{attribute 'GeneratedUsingTerminal: KL6211-0004'}
{attribute addProperty BoxType "KL6211-0004"}
{attribute addProperty Id "StatusAT %I*UINT0Parameter_InAT %I*UDINT0ASI_In_Slave_1_StatusAT %I*USINT0ASI_In_Slave_3_Slave_2AT %I*USINT0ASI_In_Slave_5_Slave_4AT %I*USINT0ASI_In_Slave_7_Slave_6AT %I*USINT0ASI_In_Slave_9_Slave_8AT %I*USINT0ASI_In_Slave_11_Slave_10AT %I*USINT0ASI_In_Slave_13_Slave_12AT %I*USINT0ASI_In_Slave_15_Slave_14AT %I*USINT0ASI_In_Slave_17_Slave_16AT %I*USINT0ASI_In_Slave_19_Slave_18AT %I*USINT0ASI_In_Slave_21_Slave_20AT %I*USINT0ASI_In_Slave_23_Slave_22AT %I*USINT0ASI_In_Slave_25_Slave_24AT %I*USINT0ASI_In_Slave_27_Slave_26AT %I*USINT0ASI_In_Slave_29_Slave_28AT %I*USINT0ASI_In_Slave_31_Slave_30AT %I*USINT0ASI_In_Slave_33_Slave_32AT %I*USINT0ASI_In_Slave_35_Slave_34AT %I*USINT0ASI_In_Slave_37_Slave_36AT %I*USINT0ASI_In_Slave_39_Slave_38AT %I*USINT0ASI_In_Slave_41_Slave_40AT %I*USINT0ASI_In_Slave_43_Slave_42AT %I*USINT0ASI_In_Slave_45_Slave_44AT %I*USINT0ASI_In_Slave_47_Slave_46AT %I*USINT0ASI_In_Slave_49_Slave_48AT %I*USINT0ASI_In_Slave_51_Slave_50AT %I*USINT0ASI_In_Slave_53_Slave_52AT %I*USINT0ASI_In_Slave_55_Slave_54AT %I*USINT0ASI_In_Slave_57_Slave_56AT %I*USINT0ASI_In_Slave_59_Slave_58AT %I*USINT0ASI_In_Slave_61_Slave_60AT %I*USINT0ASI_In_Slave_63_Slave_62AT %I*USINT0ControlAT %Q*UINT0Parameter_OutAT %Q*UDINT0ASI_Out_Slave_1_ControlAT %Q*USINT0ASI_Out_Slave_3_Slave_2AT %Q*USINT0ASI_Out_Slave_5_Slave_4AT %Q*USINT0ASI_Out_Slave_7_Slave_6AT %Q*USINT0ASI_Out_Slave_9_Slave_8AT %Q*USINT0ASI_Out_Slave_11_Slave_10AT %Q*USINT0ASI_Out_Slave_13_Slave_12AT %Q*USINT0ASI_Out_Slave_15_Slave_14AT %Q*USINT0ASI_Out_Slave_17_Slave_16AT %Q*USINT0ASI_Out_Slave_19_Slave_18AT %Q*USINT0ASI_Out_Slave_21_Slave_20AT %Q*USINT0ASI_Out_Slave_23_Slave_22AT %Q*USINT0ASI_Out_Slave_25_Slave_24AT %Q*USINT0ASI_Out_Slave_27_Slave_26AT %Q*USINT0ASI_Out_Slave_29_Slave_28AT %Q*USINT0ASI_Out_Slave_31_Slave_30AT %Q*USINT0ASI_Out_Slave_33_Slave_32AT %Q*USINT0ASI_Out_Slave_35_Slave_34AT %Q*USINT0ASI_Out_Slave_37_Slave_36AT %Q*USINT0ASI_Out_Slave_39_Slave_38AT %Q*USINT0ASI_Out_Slave_41_Slave_40AT %Q*USINT0ASI_Out_Slave_43_Slave_42AT %Q*USINT0ASI_Out_Slave_45_Slave_44AT %Q*USINT0ASI_Out_Slave_47_Slave_46AT %Q*USINT0ASI_Out_Slave_49_Slave_48AT %Q*USINT0ASI_Out_Slave_51_Slave_50AT %Q*USINT0ASI_Out_Slave_53_Slave_52AT %Q*USINT0ASI_Out_Slave_55_Slave_54AT %Q*USINT0ASI_Out_Slave_57_Slave_56AT %Q*USINT0ASI_Out_Slave_59_Slave_58AT %Q*USINT0ASI_Out_Slave_61_Slave_60AT %Q*USINT0ASI_Out_Slave_63_Slave_62AT %Q*USINT0"}
{attribute addProperty CRC "2796071749"}
{attribute addProperty Size "0"}
TYPE Channel_A6A8AB45 :
STRUCT
	{attribute addProperty Name "Status"}
	Status AT %I* : UINT;
	{attribute addProperty Name "Parameter_In"}
	Parameter_In AT %I* : UDINT;
	{attribute addProperty Name "ASI_In_Slave_1_Status"}
	ASI_In_Slave_1_Status AT %I* : USINT;
	{attribute addProperty Name "ASI_In_Slave_3_Slave_2"}
	ASI_In_Slave_3_Slave_2 AT %I* : USINT;
	{attribute addProperty Name "ASI_In_Slave_5_Slave_4"}
	ASI_In_Slave_5_Slave_4 AT %I* : USINT;
	{attribute addProperty Name "ASI_In_Slave_7_Slave_6"}
	ASI_In_Slave_7_Slave_6 AT %I* : USINT;
	{attribute addProperty Name "ASI_In_Slave_9_Slave_8"}
	ASI_In_Slave_9_Slave_8 AT %I* : USINT;
	{attribute addProperty Name "ASI_In_Slave_11_Slave_10"}
	ASI_In_Slave_11_Slave_10 AT %I* : USINT;
	{attribute addProperty Name "ASI_In_Slave_13_Slave_12"}
	ASI_In_Slave_13_Slave_12 AT %I* : USINT;
	{attribute addProperty Name "ASI_In_Slave_15_Slave_14"}
	ASI_In_Slave_15_Slave_14 AT %I* : USINT;
	{attribute addProperty Name "ASI_In_Slave_17_Slave_16"}
	ASI_In_Slave_17_Slave_16 AT %I* : USINT;
	{attribute addProperty Name "ASI_In_Slave_19_Slave_18"}
	ASI_In_Slave_19_Slave_18 AT %I* : USINT;
	{attribute addProperty Name "ASI_In_Slave_21_Slave_20"}
	ASI_In_Slave_21_Slave_20 AT %I* : USINT;
	{attribute addProperty Name "ASI_In_Slave_23_Slave_22"}
	ASI_In_Slave_23_Slave_22 AT %I* : USINT;
	{attribute addProperty Name "ASI_In_Slave_25_Slave_24"}
	ASI_In_Slave_25_Slave_24 AT %I* : USINT;
	{attribute addProperty Name "ASI_In_Slave_27_Slave_26"}
	ASI_In_Slave_27_Slave_26 AT %I* : USINT;
	{attribute addProperty Name "ASI_In_Slave_29_Slave_28"}
	ASI_In_Slave_29_Slave_28 AT %I* : USINT;
	{attribute addProperty Name "ASI_In_Slave_31_Slave_30"}
	ASI_In_Slave_31_Slave_30 AT %I* : USINT;
	{attribute addProperty Name "ASI_In_Slave_33_Slave_32"}
	ASI_In_Slave_33_Slave_32 AT %I* : USINT;
	{attribute addProperty Name "ASI_In_Slave_35_Slave_34"}
	ASI_In_Slave_35_Slave_34 AT %I* : USINT;
	{attribute addProperty Name "ASI_In_Slave_37_Slave_36"}
	ASI_In_Slave_37_Slave_36 AT %I* : USINT;
	{attribute addProperty Name "ASI_In_Slave_39_Slave_38"}
	ASI_In_Slave_39_Slave_38 AT %I* : USINT;
	{attribute addProperty Name "ASI_In_Slave_41_Slave_40"}
	ASI_In_Slave_41_Slave_40 AT %I* : USINT;
	{attribute addProperty Name "ASI_In_Slave_43_Slave_42"}
	ASI_In_Slave_43_Slave_42 AT %I* : USINT;
	{attribute addProperty Name "ASI_In_Slave_45_Slave_44"}
	ASI_In_Slave_45_Slave_44 AT %I* : USINT;
	{attribute addProperty Name "ASI_In_Slave_47_Slave_46"}
	ASI_In_Slave_47_Slave_46 AT %I* : USINT;
	{attribute addProperty Name "ASI_In_Slave_49_Slave_48"}
	ASI_In_Slave_49_Slave_48 AT %I* : USINT;
	{attribute addProperty Name "ASI_In_Slave_51_Slave_50"}
	ASI_In_Slave_51_Slave_50 AT %I* : USINT;
	{attribute addProperty Name "ASI_In_Slave_53_Slave_52"}
	ASI_In_Slave_53_Slave_52 AT %I* : USINT;
	{attribute addProperty Name "ASI_In_Slave_55_Slave_54"}
	ASI_In_Slave_55_Slave_54 AT %I* : USINT;
	{attribute addProperty Name "ASI_In_Slave_57_Slave_56"}
	ASI_In_Slave_57_Slave_56 AT %I* : USINT;
	{attribute addProperty Name "ASI_In_Slave_59_Slave_58"}
	ASI_In_Slave_59_Slave_58 AT %I* : USINT;
	{attribute addProperty Name "ASI_In_Slave_61_Slave_60"}
	ASI_In_Slave_61_Slave_60 AT %I* : USINT;
	{attribute addProperty Name "ASI_In_Slave_63_Slave_62"}
	ASI_In_Slave_63_Slave_62 AT %I* : USINT;
	{attribute addProperty Name "Control"}
	Control AT %Q* : UINT;
	{attribute addProperty Name "Parameter_Out"}
	Parameter_Out AT %Q* : UDINT;
	{attribute addProperty Name "ASI_Out_Slave_1_Control"}
	ASI_Out_Slave_1_Control AT %Q* : USINT;
	{attribute addProperty Name "ASI_Out_Slave_3_Slave_2"}
	ASI_Out_Slave_3_Slave_2 AT %Q* : USINT;
	{attribute addProperty Name "ASI_Out_Slave_5_Slave_4"}
	ASI_Out_Slave_5_Slave_4 AT %Q* : USINT;
	{attribute addProperty Name "ASI_Out_Slave_7_Slave_6"}
	ASI_Out_Slave_7_Slave_6 AT %Q* : USINT;
	{attribute addProperty Name "ASI_Out_Slave_9_Slave_8"}
	ASI_Out_Slave_9_Slave_8 AT %Q* : USINT;
	{attribute addProperty Name "ASI_Out_Slave_11_Slave_10"}
	ASI_Out_Slave_11_Slave_10 AT %Q* : USINT;
	{attribute addProperty Name "ASI_Out_Slave_13_Slave_12"}
	ASI_Out_Slave_13_Slave_12 AT %Q* : USINT;
	{attribute addProperty Name "ASI_Out_Slave_15_Slave_14"}
	ASI_Out_Slave_15_Slave_14 AT %Q* : USINT;
	{attribute addProperty Name "ASI_Out_Slave_17_Slave_16"}
	ASI_Out_Slave_17_Slave_16 AT %Q* : USINT;
	{attribute addProperty Name "ASI_Out_Slave_19_Slave_18"}
	ASI_Out_Slave_19_Slave_18 AT %Q* : USINT;
	{attribute addProperty Name "ASI_Out_Slave_21_Slave_20"}
	ASI_Out_Slave_21_Slave_20 AT %Q* : USINT;
	{attribute addProperty Name "ASI_Out_Slave_23_Slave_22"}
	ASI_Out_Slave_23_Slave_22 AT %Q* : USINT;
	{attribute addProperty Name "ASI_Out_Slave_25_Slave_24"}
	ASI_Out_Slave_25_Slave_24 AT %Q* : USINT;
	{attribute addProperty Name "ASI_Out_Slave_27_Slave_26"}
	ASI_Out_Slave_27_Slave_26 AT %Q* : USINT;
	{attribute addProperty Name "ASI_Out_Slave_29_Slave_28"}
	ASI_Out_Slave_29_Slave_28 AT %Q* : USINT;
	{attribute addProperty Name "ASI_Out_Slave_31_Slave_30"}
	ASI_Out_Slave_31_Slave_30 AT %Q* : USINT;
	{attribute addProperty Name "ASI_Out_Slave_33_Slave_32"}
	ASI_Out_Slave_33_Slave_32 AT %Q* : USINT;
	{attribute addProperty Name "ASI_Out_Slave_35_Slave_34"}
	ASI_Out_Slave_35_Slave_34 AT %Q* : USINT;
	{attribute addProperty Name "ASI_Out_Slave_37_Slave_36"}
	ASI_Out_Slave_37_Slave_36 AT %Q* : USINT;
	{attribute addProperty Name "ASI_Out_Slave_39_Slave_38"}
	ASI_Out_Slave_39_Slave_38 AT %Q* : USINT;
	{attribute addProperty Name "ASI_Out_Slave_41_Slave_40"}
	ASI_Out_Slave_41_Slave_40 AT %Q* : USINT;
	{attribute addProperty Name "ASI_Out_Slave_43_Slave_42"}
	ASI_Out_Slave_43_Slave_42 AT %Q* : USINT;
	{attribute addProperty Name "ASI_Out_Slave_45_Slave_44"}
	ASI_Out_Slave_45_Slave_44 AT %Q* : USINT;
	{attribute addProperty Name "ASI_Out_Slave_47_Slave_46"}
	ASI_Out_Slave_47_Slave_46 AT %Q* : USINT;
	{attribute addProperty Name "ASI_Out_Slave_49_Slave_48"}
	ASI_Out_Slave_49_Slave_48 AT %Q* : USINT;
	{attribute addProperty Name "ASI_Out_Slave_51_Slave_50"}
	ASI_Out_Slave_51_Slave_50 AT %Q* : USINT;
	{attribute addProperty Name "ASI_Out_Slave_53_Slave_52"}
	ASI_Out_Slave_53_Slave_52 AT %Q* : USINT;
	{attribute addProperty Name "ASI_Out_Slave_55_Slave_54"}
	ASI_Out_Slave_55_Slave_54 AT %Q* : USINT;
	{attribute addProperty Name "ASI_Out_Slave_57_Slave_56"}
	ASI_Out_Slave_57_Slave_56 AT %Q* : USINT;
	{attribute addProperty Name "ASI_Out_Slave_59_Slave_58"}
	ASI_Out_Slave_59_Slave_58 AT %Q* : USINT;
	{attribute addProperty Name "ASI_Out_Slave_61_Slave_60"}
	ASI_Out_Slave_61_Slave_60 AT %Q* : USINT;
	{attribute addProperty Name "ASI_Out_Slave_63_Slave_62"}
	ASI_Out_Slave_63_Slave_62 AT %Q* : USINT;
END_STRUCT
END_TYPE

(* stored: Version 1.2.0.0, ProductVersion 3.1.4024.9
   DUT Channel_A6A8AB45: Id {f62eeea7-df57-446f-8bec-0b393ecfab0c} *)
